# EPICS autosave request: iocs/evtIOC/iocBoot/iocEVT/auto_settings.req
file "ADEmergentVision_settings.req",  P=$(P),  R=cam1:
file "NDStdArrays_settings.req",  P=$(P),  R=image1:
file "commonPlugin_settings.req", P=$(P)
